{attribute addProperty BoxType "CU1124-0000-0016"}
{attribute addProperty Id "A_0004_CU1128_0000_0000A_0004_CU1128_0000_0000_E069C544950118.75"}
{attribute addProperty CRC "4140767130"}
{attribute addProperty SizeInBites "950"}
{attribute addProperty SizeInBytes "118.75"}
TYPE A_0003_CU1124_0000_0016_F6CF179A EXTENDS CU1124_179A0949 :
STRUCT
	{attribute addProperty Name "A_0004_CU1128_0000_0000"}
	A_0004_CU1128_0000_0000 : A_0004_CU1128_0000_0000_E069C544;
END_STRUCT
END_TYPE

(* stored: Version 1.2.0.0, ProductVersion 3.1.4024.9
   DUT A_0003_CU1124_0000_0016_F6CF179A: Id {d80b4e0e-efd6-48c2-885a-6df83a23cc32} *)
